TYPE HandlingComRequest :
STRUCT
  Start : BOOL;
  Stop : BOOL;
  GoHome : BOOL;
  Halt : BOOL;
END_STRUCT
END_TYPE

(* stored: Version 1.1.0.1
   DUT HandlingComRequest: Id {002040ed-8b7c-4996-8e3d-ba21234fe400} *)
